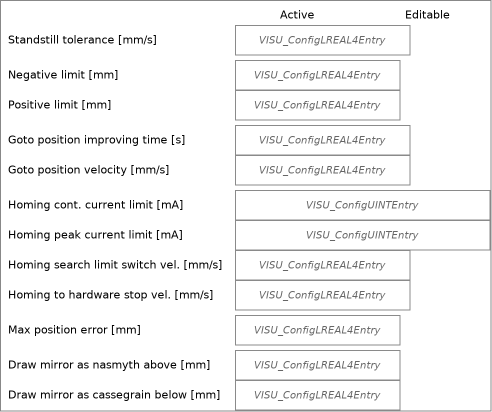
VISUALIZATION VISU_M3Config_Translation_General  // 492x412
VAR_IN_OUT
	active : M3TranslationConfig;
	editable : M3TranslationConfig;
END_VAR
    Label (235,5 125x20), "Active"
    Label (365,5 125x20), "Editable"
    Label (5,25 180x30), "Standstill tolerance [mm/s]"
    Frame (235,25 175x30)
        shows VISU_ConfigLREAL4Entry(active := active.standstillTolerance, editable := editable.standstillTolerance)
    Label (5,60 160x30), "Negative limit [mm]"
    Frame (235,60 165x30)
        shows VISU_ConfigLREAL4Entry(active := active.negativeSoftLimit, editable := editable.negativeSoftLimit)
    Frame (235,90 165x30)
        shows VISU_ConfigLREAL4Entry(active := active.positiveSoftLimit, editable := editable.positiveSoftLimit)
    Label (5,90 165x30), "Positive limit [mm]"
    Label (5,190 185x30), "Homing cont. current limit [mA]"
    Label (5,220 185x30), "Homing peak current limit [mA]"
    Frame (235,190 255x30)
        shows VISU_ConfigUINTEntry(active := active.homingContinuousCurrentLimit, editable := editable.homingContinuousCurrentLimit)
    Frame (235,220 255x30)
        shows VISU_ConfigUINTEntry(active := active.homingPeakCurrentLimit, editable := editable.homingPeakCurrentLimit)
    Label (5,250 255x30), "Homing search limit switch vel. [mm/s]"
    Frame (235,250 175x30)
        shows VISU_ConfigLREAL4Entry(active := active.homingSearchLimitSwitchVelocity, editable := editable.homingSearchLimitSwitchVelocity)
    Label (5,280 255x30), "Homing to hardware stop vel. [mm/s]"
    Frame (235,280 175x30)
        shows VISU_ConfigLREAL4Entry(active := active.homingToHardwareStopVelocity, editable := editable.homingToHardwareStopVelocity)
    Label (5,315 255x30), "Max position error [mm]"
    Frame (235,315 165x30)
        shows VISU_ConfigLREAL4Entry(active := active.maxPositionError, editable := editable.maxPositionError)
    Label (5,350 255x30), "Draw mirror as nasmyth above [mm]"
    Frame (235,350 165x30)
        shows VISU_ConfigLREAL4Entry(active := active.drawNasmythLimit, editable := editable.drawNasmythLimit)
    Label (5,380 255x30), "Draw mirror as cassegrain below [mm]"
    Frame (235,380 165x30)
        shows VISU_ConfigLREAL4Entry(active := active.drawCassegrainLimit, editable := editable.drawCassegrainLimit)
    Label (5,125 255x30), "Goto position improving time [s]"
    Frame (235,125 175x30)
        shows VISU_ConfigLREAL4Entry(active := active.gotoImprovingPositionTime, editable := editable.gotoImprovingPositionTime)
    Label (5,155 255x30), "Goto position velocity [mm/s]"
    Frame (235,155 175x30)
        shows VISU_ConfigLREAL4Entry(active := active.gotoVelocity, editable := editable.gotoVelocity)
END_VISUALIZATION

(* stored: Version 1.1.0.1, ProductVersion 3.1.4019.2
   Visu VISU_M3Config_Translation_General: Id {59c6de21-ca9a-4f1a-b3e2-ed5863171277} *)
